# EPICS autosave request: ADApp/Db/NDFileMagick_settings.req
$(P)$(R)Quality
$(P)$(R)CompressType
$(P)$(R)BitDepth
